{attribute 'linkalways'} 
{attribute 'no_explicit_call' := 'This FB is a CLASS and must be accessed using methods or properties'}
{attribute 'enable_dynamic_creation'}
FUNCTION_BLOCK Node_F_VN_FillContainer_LREAL EXTENDS VisionNode
VAR
    ipContainer : _ITcVnContainer;
    fValue : _LREAL(0.0);
    hrPrev : _HRESULT(S_OK);
    hresult : _HRESULT(S_OK);
END_VAR

METHOD PUBLIC  Clone : I_Node
VAR
    pNode : POINTER TO Node_F_VN_FillContainer_LREAL;
END_VAR
pNode := __NEW(Node_F_VN_FillContainer_LREAL);
Clone := pNode^;
END_METHOD

METHOD FB_init : BOOL
VAR_INPUT
    bInitRetains : BOOL; // if TRUE, the retain variables are initialized (warm start / cold start)
    bInCopyCode : BOOL;  // if TRUE, the instance afterwards gets moved into the copy code (online change)
END_VAR
AddInput('ipContainer', ipContainer);
AddInput('fValue', fValue);
AddInput('hrPrev', hrPrev);
AddOutput('ipContainer', ipContainer);
AddOutput('hresult',hresult);
END_METHOD

METHOD PROTECTED OnExecute : HRESULT
hresult.Value := F_VN_FillContainer_LREAL(
    ipContainer := ipContainer.Value,
    fValue := fValue.Value,
    hrPrev:= hrPrev.Value);
END_METHOD

METHOD PUBLIC PreExecutionCheck
VAR_INPUT
    Check : I_PreExecutionChecks;
END_VAR
Check.IsTrue(ipContainer.IsValid, 'ipContainer must be a valid container');
END_METHOD

END_FUNCTION_BLOCK

(* stored: Version 1.1.0.1, ProductVersion 3.1.4024.13
   POU Node_F_VN_FillContainer_LREAL: Id {5ec5ebfe-4a04-462a-a525-6efdc3bc9219}, SpecialFunc None
   Folder Constructor: Id {79415d68-ebfd-414e-bfe9-fe1179b4b2b6}
   Method Clone: Id {16b54674-5669-4289-8d66-7b9c2eb74de2}
   Method FB_init: Id {d7d5c262-b86b-49b6-b821-313e9e0ccdc8}
   Method OnExecute: Id {94d0f6b4-60ee-40fd-bdc9-b22b348ce4c9}
   Method PreExecutionCheck: Id {8043ea10-4309-4737-bcc7-52feb9e15d87} *)
